(* IEC 61131-3 sources: SigmatekTestframework/src/Class/CTestLib, 1 file *)

(* ---- CTestLib.st ---- *)
(*!
<Class
	Name               = "CTestLib"
	Revision           = "1.1"
	RealtimeTask       = "false"
	CyclicTask         = "true"
	BackgroundTask     = "true"
	DefBackground      = "10 ms"
	Sigmatek           = "false"
	OSInterface        = "false"
	HighPriority       = "false"
	Automatic          = "false"
	UpdateMode         = "Prescan"
	IconPath           = ".\Class\CTestLib\TestIcon36x36.ico"
	SharedCommandTable = "true"
	Objectsize         = "(600,420)"
	Singleton          = "true">
	<Channels>
		<Server Name="Command" Visualized="true" Initialize="true" DefValue="eCmdStop" WriteProtected="false" Retentive="false"/>
		<Server Name="eState" Visualized="true" Initialize="false" WriteProtected="true" Retentive="false"/>
		<Server Name="LastTestID" Visualized="false" Initialize="false" WriteProtected="false" Retentive="false"/>
		<Server Name="NbFailed" Visualized="true" Initialize="false" WriteProtected="true" Retentive="false"/>
		<Server Name="NbPassed" Visualized="true" Initialize="false" WriteProtected="true" Retentive="false"/>
		<Server Name="NbRun" Visualized="true" Initialize="false" WriteProtected="true" Retentive="false"/>
		<Server Name="NbSkipped" Visualized="false" Initialize="false" WriteProtected="true" Retentive="false"/>
		<Server Name="NbSuites" Visualized="true" Initialize="false" WriteProtected="true" Retentive="false"/>
		<Client Name="Classes" Required="true" Internal="false" DefValue="0"/>
		<Client Name="CodeCoverage" Required="true" Internal="true"/>
		<Client Name="JUnitReport" Required="true" Internal="true"/>
		<Client Name="Lines" Required="true" Internal="false" DefValue="0"/>
		<Client Name="LogLevel" Required="false" Internal="false" DefValue="0"/>
		<Client Name="m_strActualTest" Required="true" Internal="true"/>
		<Client Name="m_TestRunID" Required="true" Internal="true"/>
		<Client Name="m_TestSuites" Required="true" Internal="true"/>
		<Client Name="memory" Required="false" Internal="false"/>
		<Client Name="Report" Required="false" Internal="false"/>
	</Channels>
	<Dependencies>
		<Files>
			<File Path=".\Class\CTestLib\Testframework.pdf"/>
		</Files>
	</Dependencies>
	<Network Name="CTestLib">
		<!-- List of Components in this network -->
		<Components>
			<Object
				Name       = "CodeCoverage"
				Class      = "CCoverageInfo"
				Position   = "(240,810)"
				Visualized = "false">
				<Channels>
					<Server Name="Registered"/>
					<Client Name="File"/>
				</Channels>
			</Object>
			<Object
				Name       = "JUnitReport"
				Class      = "CJUnitReport"
				Position   = "(240,660)"
				Visualized = "false">
				<Channels>
					<Server Name="Registered"/>
					<Client Name="File"/>
				</Channels>
			</Object>
			<Object
				Name       = "m_strActualTest"
				Class      = "StringRAM"
				Position   = "(210,990)"
				Visualized = "true"
				Remotely   = "true">
				<Channels>
					<Server Name="Data"/>
					<Client Name="SingleRealloc" Value="1"/>
					<Client Name="UseFile"/>
				</Channels>
			</Object>
			<Object
				Name       = "m_TestRunID"
				Class      = "Ram"
				Position   = "(240,480)"
				Visualized = "true"
				Remotely   = "true">
				<Channels>
					<Server Name="Data"/>
				</Channels>
			</Object>
			<Object
				Name       = "m_TestSuites"
				Class      = "CLinkedList"
				Position   = "(210,300)"
				Visualized = "false">
				<Channels>
					<Server Name="Size"/>
					<Client Name="memory"/>
				</Channels>
			</Object>
		</Components>
		<Comments>
		</Comments>
		<!-- List of Connections in this network -->
		<Connections>
			<Connection Source="this.m_TestSuites" Destination="m_TestSuites.Size"/>
			<Connection Source="this.m_TestRunID" Destination="m_TestRunID.Data"/>
			<Connection Source="this.JUnitReport" Destination="JUnitReport.Registered"/>
			<Connection Source="this.m_strActualTest" Destination="m_strActualTest.Data"/>
			<Connection Source="this.CodeCoverage" Destination="CodeCoverage.Registered"/>
		</Connections>
		<!-- Headerfiles -->
		<Options>
		</Options>
	</Network>
</Class>
*)
CTestLib : CLASS
	TYPE
#pragma pack(push, 1)
	  SLine_t : STRUCT
	    u8Hit : USINT;
	    bBranch : BOOL;
	  END_STRUCT;
#pragma pack(pop)
	  AClassData_t : ARRAY [0..0] OF ^SLine_t;
	  ECommand_t :  //! <Type Public="true" Name="ECommand_t"/>
	  (
	    eCmdStop,
	    eCmdRun,
	    eCmdReset,
	    eCmdCreateFile
	  )$UDINT;
	  EState_t :  //! <Type Public="true" Name="EState_t"/>
	  (
	    eStateIdle,
	    eStateExecute,
	    eStateNextSuite,
	    eStateError,
	    eStateCreateJUnit,
	    eStateCreateCoverage,
	    eStateCreateReport,
	    eStateNextReport
	  )$UDINT;
	END_TYPE
  //Servers:
	eState 	: SvrChCmd_EState_t_PTofCls_CTestLib;
	LastTestID 	: SvrCh_DINT;
	NbSuites 	: SvrCh_UDINT;
	NbRun 	: SvrCh_UDINT;
	NbPassed 	: SvrCh_UDINT;
	NbFailed 	: SvrCh_UDINT;
	NbSkipped 	: SvrCh_UDINT;
	Command 	: SvrCh_ECommand_t_PTofCls_CTestLib;
  //Clients:
	m_TestSuites 	: CltChCmd_CLinkedList;
	m_TestRunID 	: CltChCmd_Ram;
	Report 	: CltChCmd_CTestReportBase;
	JUnitReport 	: CltChCmd_CJUnitReport;
	memory 	: CltChCmd_System;
	Classes 	: CltCh_UDINT;
	Lines 	: CltCh_UDINT;
	m_strActualTest 	: CltChCmd_StringRAM;
	LogLevel 	: CltCh_DINT;
	CodeCoverage 	: CltChCmd_CCoverageInfo;
  //Variables:
		m_itActSuite 	: CLinkedList::Iterator_t;
		m_udStartTime 	: UDINT;
		m_udElapsedTime 	: UDINT;
		m_pActSuite 	: ^CTestSuite;
		m_MaxIndex 	: DINT;
		m_pReport 	: ^CTestReportBase;
		m_aReports : ARRAY [0..9] OF ^CTestReportBase;

		m_u8Reports 	: USINT;
		m_u8ReportIndex 	: USINT;
		m_pClassList 	: ^UDINT;
		m_ActualTestId 	: CTestBase::ABuffer_t;
		m_pExternalTest 	: ^CExternalTest;
  //Functions:

	FUNCTION CTestLib
		VAR_OUTPUT
			ret_code 	: ConfStates;
		END_VAR;

	FUNCTION VIRTUAL GLOBAL CyWork
		VAR_INPUT
			EAX 	: UDINT;
		END_VAR
		VAR_OUTPUT
			state (EAX) 	: UDINT;
		END_VAR;

	FUNCTION VIRTUAL GLOBAL Background
		VAR_INPUT
			EAX 	: UDINT;
		END_VAR
		VAR_OUTPUT
			state (EAX) 	: UDINT;
		END_VAR;

	FUNCTION GLOBAL registerSuite
		VAR_INPUT
			pSuite 	: ^CTestSuite;
		END_VAR
		VAR_OUTPUT
			bRetcode 	: BOOL;
		END_VAR;

	FUNCTION GLOBAL getFirstTestsuite
		VAR_OUTPUT
			pFirst 	: CLinkedList::Iterator_t;
		END_VAR;

	FUNCTION GLOBAL getNextTestsuite
		VAR_INPUT
			pIterator 	: CLinkedList::Iterator_t;
		END_VAR
		VAR_OUTPUT
			pNext 	: CLinkedList::Iterator_t;
		END_VAR;

	FUNCTION GLOBAL registerReport
		VAR_INPUT
			pReport 	: ^CTestReportBase;
		END_VAR
		VAR_OUTPUT
			bRetcode 	: BOOL;
		END_VAR;

	FUNCTION GLOBAL getElement
		VAR_INPUT
			iterator 	: CLinkedList::Iterator_t;
		END_VAR
		VAR_OUTPUT
			pResult 	: ^CTestSuite;
		END_VAR;

	FUNCTION GLOBAL setActualTestId
		VAR_INPUT
			pTestId 	: ^CTestBase::ABuffer_t;
		END_VAR;

	FUNCTION InitializeMemory;

	FUNCTION Cycle;

	FUNCTION GLOBAL registerExternalTest
		VAR_INPUT
			pTest 	: ^CExternalTest;
		END_VAR
		VAR_OUTPUT
			bResult 	: DINT;
		END_VAR;
  //Tables:
	FUNCTION @STD
		VAR_OUTPUT
			ret_code	: CONFSTATES;
		END_VAR;
	FUNCTION GLOBAL TAB @CT_;
END_CLASS;

#pragma using CCoverageInfo
#pragma using CJUnitReport
#pragma using CLinkedList
#pragma using Ram
#pragma using StringRAM
#pragma usingLtd CTestReportBase
#pragma usingLtd System

#pragma usingLtd CExternalTest
#pragma usingLtd CTestReportBase
#pragma usingLtd CTestSuite

//Exclude-SccX
(*
 **********************************************************************
 * \file CTestLib.st
 *
 * Container for Testsuites
 * From here you can choose how to run your Testsuites.
 *
 * Copyright (c) 2016,Hoox.Software, Helmbrechts
 * All Rights Reserved.
 *
 * Created on: 01.06.2016
 *     Author: dressel
 *
 **********************************************************************
 *)

//*********************************************************************
//
//
//*********************************************************************
FUNCTION CTestLib::CTestLib
	VAR_OUTPUT
		ret_code 	: ConfStates;
	END_VAR

   InitializeMemory();

	ret_code := C_OK;

END_FUNCTION

//*********************************************************************
//
//
//*********************************************************************
FUNCTION GLOBAL CTestLib::registerSuite
	VAR_INPUT
		pSuite 	: ^CTestSuite;
	END_VAR
	VAR_OUTPUT
		bRetcode 	: BOOL;
	END_VAR

   bRetcode := false;

   if pSuite <> nil then

      if m_TestSuites.getElementSize() = 0 then
         m_TestSuites.create(sizeof(^CTestSuite));
      end_if;

      m_TestSuites.insert((#pSuite)$CLinkedList::ELement_t);

      NbSuites += 1;

      bRetcode := true;

   end_if;

END_FUNCTION

//*********************************************************************
//
//
//*********************************************************************
FUNCTION GLOBAL CTestLib::registerExternalTest
	VAR_INPUT
		pTest 	: ^CExternalTest;
	END_VAR
	VAR_OUTPUT
		bResult 	: DINT;
	END_VAR

   bResult := false;

   if m_pExternalTest = nil then

      m_pExternalTest := pTest;

      bResult := true;

   end_if;

END_FUNCTION

//*********************************************************************
//
//
//*********************************************************************
FUNCTION VIRTUAL GLOBAL CTestLib::Background
	VAR_INPUT
		EAX 	: UDINT;
	END_VAR
	VAR_OUTPUT
		state (EAX) 	: UDINT;
	END_VAR

   Cycle();

	state := READY;

END_FUNCTION

//*********************************************************************
//
//
//*********************************************************************
FUNCTION VIRTUAL GLOBAL CTestLib::CyWork
	VAR_INPUT
		EAX 	: UDINT;
	END_VAR
	VAR_OUTPUT
		state (EAX) 	: UDINT;
	END_VAR

   Cycle();

	State := READY;

END_FUNCTION

//*********************************************************************
//
//
//*********************************************************************
FUNCTION CTestLib::Cycle
   VAR
      sStatistic : CTestSuite::SStatistic_t;
      eReportState : CTestReportBase::ERetCode_t;
   END_VAR

   LastTestID := m_TestRunID.Data;

   m_MaxIndex := TestLib_GetSize();

   case eState of

   CTestLib::eStateIdle:

      if Command = eCmdRun then
         if m_TestSuites.empty() = false then
            m_itActSuite := m_TestSuites.first();
            m_pActSuite  := getElement(m_itActSuite);
            if m_pActSuite <> nil then
               m_pActSuite^.Prepare();
               eState       := CTestLib::eStateExecute;
               NbPassed     := 0;
               NbFailed     := 0;
               NbRun        := 0;
               NbSkipped    := 0;
               m_TestRunID.Data.Write(m_TestRunID.Data+1);
               m_udStartTime := ops.tAbsolute;
            else
               Command  := eCmdStop;
               eState   := CTestLib::eStateError;
            end_if;
         else
            if m_pExternalTest <> nil then
               m_pExternalTest^.Prepare();
               eState       := CTestLib::eStateExecute;
            else
               Command  := eCmdStop;
               eState := CTestLib::eStateError;
            end_if;

         end_if;
      end_if;

      if Command = eCmdCreateFile then
         m_u8ReportIndex := 0;
         eState          := CTestLib::eStateNextReport;
      end_if;

   CTestLib::eStateExecute:

      if m_pExternalTest <> nil then
         if m_pExternalTest^.execute() = true then
            m_pExternalTest^.cleanUp();
            eState      := eStateCreateCoverage;
         end_if;
      else

         if m_pActSuite <> nil then

            if m_pActSuite^.isSelected()  = true then

               if m_pActSuite^.execute(Command) = true then

                  eState := CTestLib::eStateNextSuite;

                  if m_pActSuite^.getStatistics(#sStatistic) = true then
                     NbRun           += sStatistic.NbRun;
                     NbPassed        += sStatistic.NbPassed;
                     NbFailed        += sStatistic.NbFailed;
                     NbSkipped       += sStatistic.NbSkipped;
                  end_if;

               end_if;

            else
               NbSkipped += 1;
               eState    := CTestLib::eStateNextSuite;

            end_if;

         else
            eState := CTestLib::eStateError;
         end_if;

      end_if;

   CTestLib::eStateNextSuite:

      m_itActSuite := m_TestSuites.next(m_itActSuite);

      if m_itActSuite <> nil then
         m_pActSuite := getElement(m_itActSuite);
         if m_pActSuite <> nil then
            m_pActSuite^.Prepare();
            eState      := CTestLib::eStateExecute;
         else
            eState      := CTestLib::eStateError;
         end_if;
      else
         m_pActSuite := nil;
         //Testlauf fertig, Testid löschen
         m_strActualTest.Clear();
         eState      := CTestLib::eStateCreateJUnit;
         Command     := eCmdStop;

         m_udElapsedTime   := ops.tAbsolute - m_udStartTime;
      end_if;

   CTestLib::eStateCreateJUnit:

      eReportState := JUnitReport.create();

      if eReportState = CTestReportBase::eFailed then
         eState   := eStateError;
      elsif eReportState = CTestReportBase::eDone then
         if m_pClassList = nil then
            eState      := eStateIdle;
            Command     := eCmdStop;
         else
            eState      := eStateCreateCoverage;
         end_if;
      end_if;

   CTestLib::eStateCreateCoverage:

      if m_pClassList <> nil then
         eReportState := CodeCoverage.create();
         if eReportState = CTestReportBase::eFailed then
            eState      := CTestLib::eStateError;
         elsif eReportState = CTestReportBase::eDone then
            eState      := CTestLib::eStateIdle;
            Command     := eCmdStop;
         end_if;
      end_if;

   CTestLib::eStateNextReport:

     m_pReport       := m_aReports[m_u8ReportIndex];
     m_u8ReportIndex +=1;
     eState          := CTestLib::eStateCreateReport;

   CTestLib::eStateCreateReport:

      if m_pReport <> nil then
         eReportState := m_pReport^.create();
      else
         eState      := CTestLib::eStateIdle;
      end_if;

      if eReportState = CTestReportBase::eFailed then
         eState   := CTestLib::eStateError;
      elsif eReportState = CTestReportBase::eDone then
         eState      := CTestLib::eStateIdle;
         Command     := eCmdStop;
      end_if;

   CTestLib::eStateError:

      if Command = eCmdReset then
         Report.reset();
         eState := CTestLib::eStateIdle;
      end_if;

   end_case;

END_FUNCTION

//*********************************************************************
//
//
//*********************************************************************
FUNCTION GLOBAL CTestLib::getFirstTestsuite
	VAR_OUTPUT
		pFirst 	: CLinkedList::Iterator_t;
	END_VAR

   pFirst := m_TestSuites.first();

END_FUNCTION

//*********************************************************************
//
//
//*********************************************************************
FUNCTION GLOBAL CTestLib::getNextTestsuite
	VAR_INPUT
		pIterator 	: CLinkedList::Iterator_t;
	END_VAR
	VAR_OUTPUT
		pNext 	: CLinkedList::Iterator_t;
	END_VAR

   pNext := m_TestSuites.next(pIterator);

END_FUNCTION

//*********************************************************************
//
//
//*********************************************************************
FUNCTION GLOBAL CTestLib::registerReport
	VAR_INPUT
		pReport 	: ^CTestreportBase;
	END_VAR
	VAR_OUTPUT
		bRetcode 	: BOOL;
	END_VAR

   bRetcode    := false;

   if pReport = nil then
      return;
   end_if;
   // interne Elemente nicht registrieren
   if JUnitReport.compare(pReport) then
      return;
   end_if;

   if m_u8Reports = 9 then
      return;
   end_if;

   m_aReports[m_u8Reports] := pReport;
   m_u8Reports += 1;

END_FUNCTION

//*********************************************************************
//
//
//*********************************************************************
FUNCTION GLOBAL CTestLib::getElement
	VAR_INPUT
		iterator 	: CLinkedList::Iterator_t;
	END_VAR
	VAR_OUTPUT
		pResult 	: ^CTestSuite;
	END_VAR

   m_TestSuites.getElement(iterator , (#pResult)$CLinkedList::Element_t);

END_FUNCTION

//*********************************************************************
//
//
//*********************************************************************
FUNCTION GLOBAL CTestLib::setActualTestId
	VAR_INPUT
		pTestId 	: ^CTestBase::ABuffer_t;
	END_VAR

   if pTestId = nil then
      return;
   end_if;

   memory.MemSet(pMemptr   := #m_ActualTestId,
                 fill      := 0,
                 size      := sizeof(CTestBase::ABuffer_t));

   memory.MemCpy( dest     := #m_ActualTestId,
                  source   := pTestId,
                  size     := sizeof(CTestBase::ABuffer_t));

   m_strActualTest.Clear();
   m_strActualTest.WriteDataOff(udLen:= _StrLen(src:= #m_ActualTestId[0]),
                                udOff:= 0,
                                pData:= #m_ActualTestId[0]);

END_FUNCTION

//*********************************************************************
//
//
//*********************************************************************
FUNCTION CTestLib::InitializeMemory
VAR
	u32Index  : UDINT;
   pClass    : ^UDINT;
   pLineInfo : ^void;
   u32Size   : UDINT;
END_VAR

   Command := eCmdStop;

   if Classes > 0 then
      u32Size := Classes*sizeof(AClassData_t);
      // Speicher für Klassenliste reservieren
      m_pClassList$^void := memory.Malloc(u32Size);
      if (m_pClassList <> nil) then
         memory.MemSet(m_pClassList, 0, u32Size);
      end_if;

      if m_pClassList = nil then
         TRACE_ERR("InitializeMemory failed to create Classlist!");
         eState := CTestLib::EStateError;
         return;
      end_if;

      pClass  := m_pClassList;
      u32Size := Lines*sizeof(SLine_t);
      // Speicher für Zeilen in den Klassen reservieren
      for u32Index := 0 to Classes-1 do
         pLineInfo := memory.Malloc(u32Size);

         if (pLineInfo <> nil) then
            memory.MemSet(pLineInfo, 0, u32Size);
            pClass^ := pLineInfo$UDINT;
         else
            TRACE_ERR("InitializeMemory failed to create Line Memory!");
            eState   := CTestLib::EStateError;
            u32Index := Classes;
         end_if;

         pClass  += sizeof(UDINT);
      end_for;

      TestLib_Init(m_pClassList, Classes, Lines);
   end_if;

END_FUNCTION
